// TIA Portal V20 export
DATA_BLOCK "PNDevDiagStatus"   // DB231
// stored: InstanceOfName LER_DiagnosticsInterface, InstanceOfType UDT
"LER_DiagnosticsInterface"
   // VAR
   //    DevState { S7_SetPoint := 'True'} : "LER_DevState";
   //    DigState { S7_SetPoint := 'True'} : Array[0..15] of Bool;
   //    Station_Position : Int := 0;
   // END_VAR
BEGIN
   DevState.DevState_X1.staticDevState1[0..100].devNumber := 0;
   DevState.DevState_X1.staticDevState1[0..100].devName := '';
   DevState.DevState_X1.staticDevState1[0..100].devStateDezCoded := 0;
   DevState.DevState_X1.staticDevState1[0..100].devStateBitCoded := 16#0000;
   DevState.DevState_X1.staticDevState1[0..100].first8CharOfMlfb := '';
   DevState.DevState_X1.staticDevState2[0..100].devNumber := 0;
   DevState.DevState_X1.staticDevState2[0..100].devName := '';
   DevState.DevState_X1.staticDevState2[0..100].devStateDezCoded := 0;
   DevState.DevState_X1.staticDevState2[0..100].devStateBitCoded := 16#0000;
   DevState.DevState_X1.staticDevState2[0..100].first8CharOfMlfb := '';
   DevState.DevState_X1.staticDevState3[0..100].devNumber := 0;
   DevState.DevState_X1.staticDevState3[0..100].devName := '';
   DevState.DevState_X1.staticDevState3[0..100].devStateDezCoded := 0;
   DevState.DevState_X1.staticDevState3[0..100].devStateBitCoded := 16#0000;
   DevState.DevState_X1.staticDevState3[0..100].first8CharOfMlfb := '';
   DevState.DevState_X1.staticDevState4[0..100].devNumber := 0;
   DevState.DevState_X1.staticDevState4[0..100].devName := '';
   DevState.DevState_X1.staticDevState4[0..100].devStateDezCoded := 0;
   DevState.DevState_X1.staticDevState4[0..100].devStateBitCoded := 16#0000;
   DevState.DevState_X1.staticDevState4[0..100].first8CharOfMlfb := '';
   DevState.DevState_X1.staticDevState5[0..100].devNumber := 0;
   DevState.DevState_X1.staticDevState5[0..100].devName := '';
   DevState.DevState_X1.staticDevState5[0..100].devStateDezCoded := 0;
   DevState.DevState_X1.staticDevState5[0..100].devStateBitCoded := 16#0000;
   DevState.DevState_X1.staticDevState5[0..100].first8CharOfMlfb := '';
   DevState.DevState_X1.staticDevState6[0..100].devNumber := 0;
   DevState.DevState_X1.staticDevState6[0..100].devName := '';
   DevState.DevState_X1.staticDevState6[0..100].devStateDezCoded := 0;
   DevState.DevState_X1.staticDevState6[0..100].devStateBitCoded := 16#0000;
   DevState.DevState_X1.staticDevState6[0..100].first8CharOfMlfb := '';
   DevState.DevState_X1.staticDevState7[0..100].devNumber := 0;
   DevState.DevState_X1.staticDevState7[0..100].devName := '';
   DevState.DevState_X1.staticDevState7[0..100].devStateDezCoded := 0;
   DevState.DevState_X1.staticDevState7[0..100].devStateBitCoded := 16#0000;
   DevState.DevState_X1.staticDevState7[0..100].first8CharOfMlfb := '';
   DevState.DevState_X1.staticDevState8[0..100].devNumber := 0;
   DevState.DevState_X1.staticDevState8[0..100].devName := '';
   DevState.DevState_X1.staticDevState8[0..100].devStateDezCoded := 0;
   DevState.DevState_X1.staticDevState8[0..100].devStateBitCoded := 16#0000;
   DevState.DevState_X1.staticDevState8[0..100].first8CharOfMlfb := '';
   DevState.DevState_X1.staticDevState9[0..100].devNumber := 0;
   DevState.DevState_X1.staticDevState9[0..100].devName := '';
   DevState.DevState_X1.staticDevState9[0..100].devStateDezCoded := 0;
   DevState.DevState_X1.staticDevState9[0..100].devStateBitCoded := 16#0000;
   DevState.DevState_X1.staticDevState9[0..100].first8CharOfMlfb := '';
   DevState.DevState_X1.staticDevState10[0..100].devNumber := 0;
   DevState.DevState_X1.staticDevState10[0..100].devName := '';
   DevState.DevState_X1.staticDevState10[0..100].devStateDezCoded := 0;
   DevState.DevState_X1.staticDevState10[0..100].devStateBitCoded := 16#0000;
   DevState.DevState_X1.staticDevState10[0..100].first8CharOfMlfb := '';
   DevState.DevState_X1.staticDevState11[0..100].devNumber := 0;
   DevState.DevState_X1.staticDevState11[0..100].devName := '';
   DevState.DevState_X1.staticDevState11[0..100].devStateDezCoded := 0;
   DevState.DevState_X1.staticDevState11[0..100].devStateBitCoded := 16#0000;
   DevState.DevState_X1.staticDevState11[0..100].first8CharOfMlfb := '';
   DevState.DevState_X1.staticDevState12[0..100].devNumber := 0;
   DevState.DevState_X1.staticDevState12[0..100].devName := '';
   DevState.DevState_X1.staticDevState12[0..100].devStateDezCoded := 0;
   DevState.DevState_X1.staticDevState12[0..100].devStateBitCoded := 16#0000;
   DevState.DevState_X1.staticDevState12[0..100].first8CharOfMlfb := '';
   DevState.DevState_X1.staticDevState13[0..100].devNumber := 0;
   DevState.DevState_X1.staticDevState13[0..100].devName := '';
   DevState.DevState_X1.staticDevState13[0..100].devStateDezCoded := 0;
   DevState.DevState_X1.staticDevState13[0..100].devStateBitCoded := 16#0000;
   DevState.DevState_X1.staticDevState13[0..100].first8CharOfMlfb := '';
   DevState.DevState_X1.staticDevState14[0..100].devNumber := 0;
   DevState.DevState_X1.staticDevState14[0..100].devName := '';
   DevState.DevState_X1.staticDevState14[0..100].devStateDezCoded := 0;
   DevState.DevState_X1.staticDevState14[0..100].devStateBitCoded := 16#0000;
   DevState.DevState_X1.staticDevState14[0..100].first8CharOfMlfb := '';
   DevState.DevState_X1.staticDevState15[0..100].devNumber := 0;
   DevState.DevState_X1.staticDevState15[0..100].devName := '';
   DevState.DevState_X1.staticDevState15[0..100].devStateDezCoded := 0;
   DevState.DevState_X1.staticDevState15[0..100].devStateBitCoded := 16#0000;
   DevState.DevState_X1.staticDevState15[0..100].first8CharOfMlfb := '';
   DevState.DevState_X2.staticDevState1[0..100].devNumber := 0;
   DevState.DevState_X2.staticDevState1[0..100].devName := '';
   DevState.DevState_X2.staticDevState1[0..100].devStateDezCoded := 0;
   DevState.DevState_X2.staticDevState1[0..100].devStateBitCoded := 16#0000;
   DevState.DevState_X2.staticDevState1[0..100].first8CharOfMlfb := '';
   DevState.DevState_X2.staticDevState2[0..100].devNumber := 0;
   DevState.DevState_X2.staticDevState2[0..100].devName := '';
   DevState.DevState_X2.staticDevState2[0..100].devStateDezCoded := 0;
   DevState.DevState_X2.staticDevState2[0..100].devStateBitCoded := 16#0000;
   DevState.DevState_X2.staticDevState2[0..100].first8CharOfMlfb := '';
   DevState.DevState_X2.staticDevState3[0..100].devNumber := 0;
   DevState.DevState_X2.staticDevState3[0..100].devName := '';
   DevState.DevState_X2.staticDevState3[0..100].devStateDezCoded := 0;
   DevState.DevState_X2.staticDevState3[0..100].devStateBitCoded := 16#0000;
   DevState.DevState_X2.staticDevState3[0..100].first8CharOfMlfb := '';
   DevState.DevState_X2.staticDevState4[0..100].devNumber := 0;
   DevState.DevState_X2.staticDevState4[0..100].devName := '';
   DevState.DevState_X2.staticDevState4[0..100].devStateDezCoded := 0;
   DevState.DevState_X2.staticDevState4[0..100].devStateBitCoded := 16#0000;
   DevState.DevState_X2.staticDevState4[0..100].first8CharOfMlfb := '';
   DevState.DevState_X2.staticDevState5[0..100].devNumber := 0;
   DevState.DevState_X2.staticDevState5[0..100].devName := '';
   DevState.DevState_X2.staticDevState5[0..100].devStateDezCoded := 0;
   DevState.DevState_X2.staticDevState5[0..100].devStateBitCoded := 16#0000;
   DevState.DevState_X2.staticDevState5[0..100].first8CharOfMlfb := '';
   DevState.DevState_X2.staticDevState6[0..100].devNumber := 0;
   DevState.DevState_X2.staticDevState6[0..100].devName := '';
   DevState.DevState_X2.staticDevState6[0..100].devStateDezCoded := 0;
   DevState.DevState_X2.staticDevState6[0..100].devStateBitCoded := 16#0000;
   DevState.DevState_X2.staticDevState6[0..100].first8CharOfMlfb := '';
   DevState.DevState_X2.staticDevState7[0..100].devNumber := 0;
   DevState.DevState_X2.staticDevState7[0..100].devName := '';
   DevState.DevState_X2.staticDevState7[0..100].devStateDezCoded := 0;
   DevState.DevState_X2.staticDevState7[0..100].devStateBitCoded := 16#0000;
   DevState.DevState_X2.staticDevState7[0..100].first8CharOfMlfb := '';
   DevState.DevState_X2.staticDevState8[0..100].devNumber := 0;
   DevState.DevState_X2.staticDevState8[0..100].devName := '';
   DevState.DevState_X2.staticDevState8[0..100].devStateDezCoded := 0;
   DevState.DevState_X2.staticDevState8[0..100].devStateBitCoded := 16#0000;
   DevState.DevState_X2.staticDevState8[0..100].first8CharOfMlfb := '';
   DevState.DevState_X2.staticDevState9[0..100].devNumber := 0;
   DevState.DevState_X2.staticDevState9[0..100].devName := '';
   DevState.DevState_X2.staticDevState9[0..100].devStateDezCoded := 0;
   DevState.DevState_X2.staticDevState9[0..100].devStateBitCoded := 16#0000;
   DevState.DevState_X2.staticDevState9[0..100].first8CharOfMlfb := '';
   DevState.DevState_X2.staticDevState10[0..100].devNumber := 0;
   DevState.DevState_X2.staticDevState10[0..100].devName := '';
   DevState.DevState_X2.staticDevState10[0..100].devStateDezCoded := 0;
   DevState.DevState_X2.staticDevState10[0..100].devStateBitCoded := 16#0000;
   DevState.DevState_X2.staticDevState10[0..100].first8CharOfMlfb := '';
   DevState.DevState_X2.staticDevState11[0..100].devNumber := 0;
   DevState.DevState_X2.staticDevState11[0..100].devName := '';
   DevState.DevState_X2.staticDevState11[0..100].devStateDezCoded := 0;
   DevState.DevState_X2.staticDevState11[0..100].devStateBitCoded := 16#0000;
   DevState.DevState_X2.staticDevState11[0..100].first8CharOfMlfb := '';
   DevState.DevState_X2.staticDevState12[0..100].devNumber := 0;
   DevState.DevState_X2.staticDevState12[0..100].devName := '';
   DevState.DevState_X2.staticDevState12[0..100].devStateDezCoded := 0;
   DevState.DevState_X2.staticDevState12[0..100].devStateBitCoded := 16#0000;
   DevState.DevState_X2.staticDevState12[0..100].first8CharOfMlfb := '';
   DevState.DevState_X2.staticDevState13[0..100].devNumber := 0;
   DevState.DevState_X2.staticDevState13[0..100].devName := '';
   DevState.DevState_X2.staticDevState13[0..100].devStateDezCoded := 0;
   DevState.DevState_X2.staticDevState13[0..100].devStateBitCoded := 16#0000;
   DevState.DevState_X2.staticDevState13[0..100].first8CharOfMlfb := '';
   DevState.DevState_X2.staticDevState14[0..100].devNumber := 0;
   DevState.DevState_X2.staticDevState14[0..100].devName := '';
   DevState.DevState_X2.staticDevState14[0..100].devStateDezCoded := 0;
   DevState.DevState_X2.staticDevState14[0..100].devStateBitCoded := 16#0000;
   DevState.DevState_X2.staticDevState14[0..100].first8CharOfMlfb := '';
   DevState.DevState_X2.staticDevState15[0..100].devNumber := 0;
   DevState.DevState_X2.staticDevState15[0..100].devName := '';
   DevState.DevState_X2.staticDevState15[0..100].devStateDezCoded := 0;
   DevState.DevState_X2.staticDevState15[0..100].devStateBitCoded := 16#0000;
   DevState.DevState_X2.staticDevState15[0..100].first8CharOfMlfb := '';
   DevState.DevState.staticDevState1[0..100].devNumber := 0;
   DevState.DevState.staticDevState1[0..100].devName := '';
   DevState.DevState.staticDevState1[0..100].devStateDezCoded := 0;
   DevState.DevState.staticDevState1[0..100].devStateBitCoded := 16#0000;
   DevState.DevState.staticDevState1[0..100].first8CharOfMlfb := '';
   DevState.DevState.staticDevState2[0..100].devNumber := 0;
   DevState.DevState.staticDevState2[0..100].devName := '';
   DevState.DevState.staticDevState2[0..100].devStateDezCoded := 0;
   DevState.DevState.staticDevState2[0..100].devStateBitCoded := 16#0000;
   DevState.DevState.staticDevState2[0..100].first8CharOfMlfb := '';
   DevState.DevState.staticDevState3[0..100].devNumber := 0;
   DevState.DevState.staticDevState3[0..100].devName := '';
   DevState.DevState.staticDevState3[0..100].devStateDezCoded := 0;
   DevState.DevState.staticDevState3[0..100].devStateBitCoded := 16#0000;
   DevState.DevState.staticDevState3[0..100].first8CharOfMlfb := '';
   DevState.DevState.staticDevState4[0..100].devNumber := 0;
   DevState.DevState.staticDevState4[0..100].devName := '';
   DevState.DevState.staticDevState4[0..100].devStateDezCoded := 0;
   DevState.DevState.staticDevState4[0..100].devStateBitCoded := 16#0000;
   DevState.DevState.staticDevState4[0..100].first8CharOfMlfb := '';
   DevState.DevState.staticDevState5[0..100].devNumber := 0;
   DevState.DevState.staticDevState5[0..100].devName := '';
   DevState.DevState.staticDevState5[0..100].devStateDezCoded := 0;
   DevState.DevState.staticDevState5[0..100].devStateBitCoded := 16#0000;
   DevState.DevState.staticDevState5[0..100].first8CharOfMlfb := '';
   DevState.DevState.staticDevState6[0..100].devNumber := 0;
   DevState.DevState.staticDevState6[0..100].devName := '';
   DevState.DevState.staticDevState6[0..100].devStateDezCoded := 0;
   DevState.DevState.staticDevState6[0..100].devStateBitCoded := 16#0000;
   DevState.DevState.staticDevState6[0..100].first8CharOfMlfb := '';
   DevState.DevState.staticDevState7[0..100].devNumber := 0;
   DevState.DevState.staticDevState7[0..100].devName := '';
   DevState.DevState.staticDevState7[0..100].devStateDezCoded := 0;
   DevState.DevState.staticDevState7[0..100].devStateBitCoded := 16#0000;
   DevState.DevState.staticDevState7[0..100].first8CharOfMlfb := '';
   DevState.DevState.staticDevState8[0..100].devNumber := 0;
   DevState.DevState.staticDevState8[0..100].devName := '';
   DevState.DevState.staticDevState8[0..100].devStateDezCoded := 0;
   DevState.DevState.staticDevState8[0..100].devStateBitCoded := 16#0000;
   DevState.DevState.staticDevState8[0..100].first8CharOfMlfb := '';
   DevState.DevState.staticDevState9[0..100].devNumber := 0;
   DevState.DevState.staticDevState9[0..100].devName := '';
   DevState.DevState.staticDevState9[0..100].devStateDezCoded := 0;
   DevState.DevState.staticDevState9[0..100].devStateBitCoded := 16#0000;
   DevState.DevState.staticDevState9[0..100].first8CharOfMlfb := '';
   DevState.DevState.staticDevState10[0..100].devNumber := 0;
   DevState.DevState.staticDevState10[0..100].devName := '';
   DevState.DevState.staticDevState10[0..100].devStateDezCoded := 0;
   DevState.DevState.staticDevState10[0..100].devStateBitCoded := 16#0000;
   DevState.DevState.staticDevState10[0..100].first8CharOfMlfb := '';
   DevState.DevState.staticDevState11[0..100].devNumber := 0;
   DevState.DevState.staticDevState11[0..100].devName := '';
   DevState.DevState.staticDevState11[0..100].devStateDezCoded := 0;
   DevState.DevState.staticDevState11[0..100].devStateBitCoded := 16#0000;
   DevState.DevState.staticDevState11[0..100].first8CharOfMlfb := '';
   DevState.DevState.staticDevState12[0..100].devNumber := 0;
   DevState.DevState.staticDevState12[0..100].devName := '';
   DevState.DevState.staticDevState12[0..100].devStateDezCoded := 0;
   DevState.DevState.staticDevState12[0..100].devStateBitCoded := 16#0000;
   DevState.DevState.staticDevState12[0..100].first8CharOfMlfb := '';
   DevState.DevState.staticDevState13[0..100].devNumber := 0;
   DevState.DevState.staticDevState13[0..100].devName := '';
   DevState.DevState.staticDevState13[0..100].devStateDezCoded := 0;
   DevState.DevState.staticDevState13[0..100].devStateBitCoded := 16#0000;
   DevState.DevState.staticDevState13[0..100].first8CharOfMlfb := '';
   DevState.DevState.staticDevState14[0..100].devNumber := 0;
   DevState.DevState.staticDevState14[0..100].devName := '';
   DevState.DevState.staticDevState14[0..100].devStateDezCoded := 0;
   DevState.DevState.staticDevState14[0..100].devStateBitCoded := 16#0000;
   DevState.DevState.staticDevState14[0..100].first8CharOfMlfb := '';
   DevState.DevState.staticDevState15[0..100].devNumber := 0;
   DevState.DevState.staticDevState15[0..100].devName := '';
   DevState.DevState.staticDevState15[0..100].devStateDezCoded := 0;
   DevState.DevState.staticDevState15[0..100].devStateBitCoded := 16#0000;
   DevState.DevState.staticDevState15[0..100].first8CharOfMlfb := '';
   DigState[0] := FALSE;
   DigState[1..9] := TRUE;
   DigState[10..15] := FALSE;
END_DATA_BLOCK
